FUNCTION Convert_SINT_TO_DT : BOOL
VAR_INPUT
	in : SINT;
	out : REFERENCE TO DT;
END_VAR
VAR
	converted : DT;
END_VAR

converted := SINT_TO_DT(in);

IF (DT_TO_SINT(converted) <> in) THEN
	RETURN;
END_IF

out := converted;
Convert_SINT_TO_DT := TRUE;

END_FUNCTION

(* stored: Version 1.1.0.1, ProductVersion 3.1.4024.12
   POU Convert_SINT_TO_DT: Id {6508de79-bd33-494d-9c04-e03ffe7540a2}, SpecialFunc None *)
